Fanuc KAREL source: ko00040.KL

-- PROVISIONAL review KL for V770-1; original PC SHA256 6c1339938a93aba14ad2d87989db271076cac1018c30a7ef09791c8716ca61cd
-- Incomplete behavior may be omitted. Consult companion uncertainty JSON. Do not deploy.
PROGRAM KO00040
%NOLOCKGROUP
BEGIN
  -- UNRESOLVED_PC offsets 5-12; opcodes 9D,23
  -- UNRESOLVED_PC offsets 17-69; opcodes 27,27,49,7E,AD,27,49,7E,AD,22,31,7E,4A
  -- UNRESOLVED_PC offsets 74-78; opcodes 7F
END KO00040
